FUNCTION_BLOCK FB_StopWatch
VAR_INPUT
	bStart: BOOL;
	bReset: BOOL;
END_VAR
VAR_IN_OUT
	tElapsedTime: TIME;
END_VAR
VAR
	tStartTime: TIME;
	rtReset: R_TRIG;
	tLastElapsedTime: TIME;
END_VAR

rtReset(CLK:= bReset);
IF rtReset.Q THEN
	F_Clear(tLastElapsedTime);
	F_Clear(tStartTime);
END_IF

IF bStart AND tStartTime = T#0MS THEN
	tStartTime:= TIME();
ELSIF NOT bStart AND tStartTime > T#0MS THEN
	tLastElapsedTime:= tLastElapsedTime + TIME() - tStartTime;
	F_Clear(tStartTime);
END_IF

IF tStartTime > T#0MS THEN
	tElapsedTime:= tLastElapsedTime + TIME() - tStartTime;
ELSIF tLastElapsedTime = T#0S AND tElapsedTime > T#0S THEN
	tLastElapsedTime:= tElapsedTime;
ELSE
	tElapsedTime:= tLastElapsedTime;
END_IF

END_FUNCTION_BLOCK

(* stored: Version 1.1.0.1, ProductVersion 3.1.4024.12
   POU FB_StopWatch: Id {10b17d02-3164-4219-9e87-e977ce578348}, SpecialFunc None *)
